FUNCTION_BLOCK FB_Mirror_States EXTENDS FB_PositionStateBase_WithPMPS
VAR_INPUT
    enumSet: INT;
    stMR1In: DUT_PositionState;
    stMR1Out: DUT_PositionState;
    
END_VAR
VAR_OUTPUT
END_VAR
VAR
END_VAR

END_FUNCTION_BLOCK

(* stored: Version 1.1.0.1, ProductVersion 3.1.4022.18
   POU FB_Mirror_States: Id {f73817f2-6bf1-4d67-937c-f4841113134d}, SpecialFunc None *)
